// TIA Portal V18 export
// export: Created 2026-06-08T16:08:50.0383366Z, ExportSetting WithDefaults, DisplayName Totally Integrated Automation Portal, DisplayVersion V18, DisplayName TIA Portal Openness, DisplayVersion V18, DisplayName TIA Portal Version Control Interface, DisplayVersion V18, DisplayName STEP 7 Professional, DisplayVersion V18, DisplayName STEP 7 Safety, DisplayVersion V18, DisplayName WinCC Professional, DisplayVersion V18
FUNCTION "FC_MO_PHONG_ND" : Void   // FC1, LAD
{ S7_Optimized_Access := 'TRUE' }
VERSION : 0.1
// stored: AutoNumber true, IsIECCheckEnabled false, SetENOAutomatically false, UDAEnableTagReadback false
   VAR_TEMP   // added for the SCL form of the ladder/FBD networks
      _w1 : Bool;
      _w2 : Bool;
      _w3 : Bool;
      _w4 : Bool;
   END_VAR
BEGIN

REGION Network 1
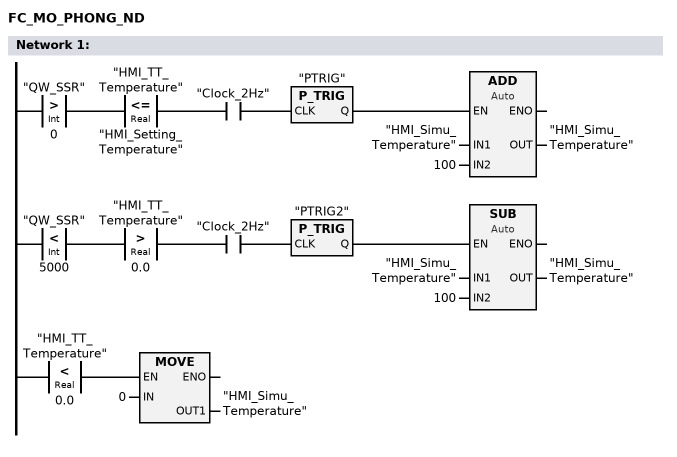
   RUNG wire#powerrail
      { S7_Templates := "SrcType := Int" } GT_Contact(in1 := "QW_SSR", in2 := 0)
      { S7_Templates := "SrcType := Real" } LE_Contact(in1 := "HMI_TT_Temperature", in2 := "HMI_Setting_Temperature")
      Contact( "Clock_2Hz" )
      P_Trig( "PTRIG" )
      Add(in1 := "HMI_Simu_Temperature", in2 := 100, out => "HMI_Simu_Temperature")
   END_RUNG
   RUNG wire#powerrail
      { S7_Templates := "SrcType := Int" } LT_Contact(in1 := "QW_SSR", in2 := 5000)
      { S7_Templates := "SrcType := Real" } GT_Contact(in1 := "HMI_TT_Temperature", in2 := 0.0)
      Contact( "Clock_2Hz" )
      P_Trig( "PTRIG2" )
      Sub(in1 := "HMI_Simu_Temperature", in2 := 100, out => "HMI_Simu_Temperature")
   END_RUNG
   RUNG wire#powerrail
      { S7_Templates := "SrcType := Real" } LT_Contact(in1 := "HMI_TT_Temperature", in2 := 0.0)
      Move(in := 0, out1 => "HMI_Simu_Temperature")
   END_RUNG
   // the same network as SCL:
   #_w1 := ("QW_SSR" > 0) AND ("HMI_TT_Temperature" <= "HMI_Setting_Temperature") AND "Clock_2Hz";
   #_w2 := #_w1 AND NOT "PTRIG";   // rising edge
   "PTRIG" := #_w1;
   IF #_w2 THEN "HMI_Simu_Temperature" := "HMI_Simu_Temperature" + 100; END_IF;
   #_w3 := ("QW_SSR" < 5000) AND ("HMI_TT_Temperature" > 0.0) AND "Clock_2Hz";
   #_w4 := #_w3 AND NOT "PTRIG2";   // rising edge
   "PTRIG2" := #_w3;
   IF #_w4 THEN "HMI_Simu_Temperature" := "HMI_Simu_Temperature" - 100; END_IF;
   IF "HMI_TT_Temperature" < 0.0 THEN "HMI_Simu_Temperature" := 0; END_IF;
END_REGION
END_FUNCTION
